// Mitsubishi GX Works2 project: mcEx03   PLC: Q02/Q02H

PROGRAM MAIN
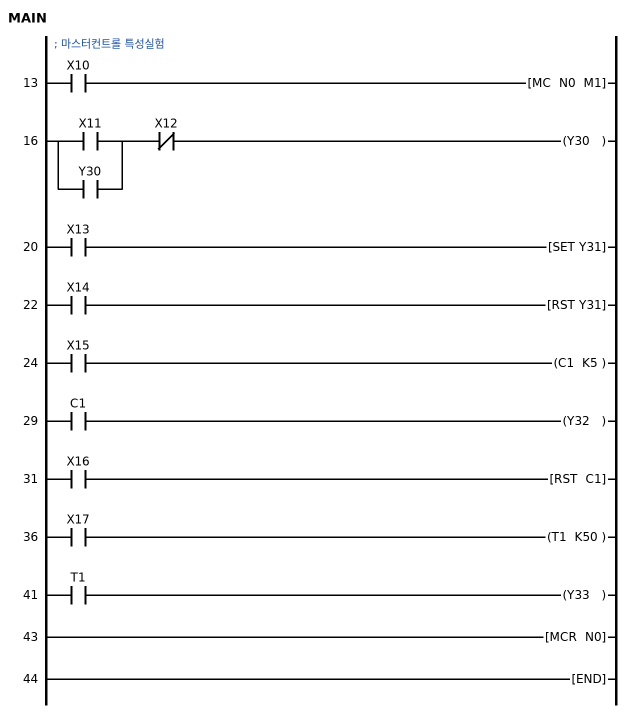
; 마스터컨트롤 특성실험
13    LD      X10
      MC      N0 M1
16    LD      X11
      OR      Y30
      ANI     X12
      OUT     Y30
20    LD      X13
      SET     Y31
22    LD      X14
      RST     Y31
24    LD      X15
      OUT     C1 K5
29    LD      C1
      OUT     Y32
31    LD      X16
      RST     C1
36    LD      X17
      OUT     T1 K50
41    LD      T1
      OUT     Y33
43    MCR     N0
44    END
END_PROGRAM
